Staubli VAL3: Welcome.dtx

mdesc mNomSpeed
